FUNCTION_BLOCK Axis
//VAR_INPUT	
//END_VAR
VAR_OUTPUT
	Axis_Error			: BOOL;				// Error signal
	Axis_ErrorID		: UDINT;			// Error ID
	Axis_Moves			: BOOL;				// Status of moving
END_VAR
VAR
	// =============== Done signals MC Block =================
	JogDone			    : BOOL;					// Status of function block MC_Jog
	ResetDone		    : BOOL;					// Status of function block MC_Reset
	HaltDone		    : BOOL;					// Status of function block MC_Halt
	HomeDone		    : BOOL;					// Status of function block MC_Home
  	MoveAbsoluteDone : BOOL;        // Status of function block MC_MoveAbsolute
  	ExtSetPiontDone 	: BOOL;         		// Status of function block MC_ExtSetPointGenDisable

	// =============== Control variables ======================
	//Home_Back_Start	: BOOL;
	//Drive_Home		: BOOL;
	
	// =============== State variables ========================
	Power_StatusEnable	: BOOL;					// Enable feedback
	
	// ============= Velocity, override ,Position==============
	Velocity_Jog		: LREAL;				// Jog velocity
	Velocity_Move		: LREAL;				// Target velocity
	Velocity_Home		: LREAL;				// Home velocity
	Velocity_Absolute	: LREAL;				// MoveAbsolute velocity
	Velocity_Relative	: LREAL;				// MoveRelative velocity
	fOverride 			: LREAL := 100.0;		// Override 100%
  Home_Position   : LREAL;        // The absolute position after Home will be
	
	// =============== Trigger function blocks ================
	
	TriggerHalt	: R_TRIG;				// Trigger to recognize rising edge of halt input
	TriggerReset : R_TRIG;				// Trigger to recognize rising edge of reset input
	
	// =============== Axis reference =========================
	AxisRef			: AXIS_REF;				// Axis reference (process data plc/nc)
	
	// =============== About axis turque ====================
	Axis_Current_Turque 	: INT;
  	Axis_Max_Turque       	: INT;

	// ================= Sensor FeedBack ====================
  	Proximity_Switch      : DINT;
	
	// =============== Motion function blocks =================
	Axis_Power 			: MC_Power;				// FB for enable and override			[上电]
	Axis_Home			: MC_Home;				// FB for axis home						[找零]
	Axis_Reset 			: MC_Reset;				// FB to reset axis						[复位]
	Axis_Jog			: MC_Jog;				// FB to jog axis						[点动]
	Axis_Stop 			: MC_Stop;				// FB to stop axis						[停止]
	Axis_Halt			: MC_Halt;				// FB to halt axis						[停止]
	Axis_Move			: MC_MoveVelocity;		// FB to move axis (velocity movement)	[匀速运动]
	Axis_MoveAbsolute 	: MC_MoveAbsolute;		// FB to move axis absolutely			[绝对位置运动]
	Axis_MoveRelative	: MC_MoveRelative;		// FB to move axis relatively			[相对位置运动]
  	Axis_ActPosition  : MC_ReadActualPosition; // FB to read the actual position of axis  [读取电机轴的实际位置]
	Axis_ActVelocity	: MC_ReadActualVelocity;// FB to read the actual Velocity of axis [读取电机轴的实际速度]
	Axis_Delay			: Delay;				// FB to operate the delay program		[延迟程序]
	Axis_ExtSetPiontEnable	: MC_ExtSetPointGenEnable;	// FB to enable extsetpoint		[外部函数发生使能]
	Axis_ExtSetPiontDisable	: MC_ExtSetPointGenDisable;	// FB to disable extsetpoint	[外部函数结束使能]
  
  // =============== Timer =================
  Delay         : TON;          //[定时器]
END_VAR

PROPERTY ActPosition : LREAL
GET
Axis_ActPosition( Axis:= AxisRef, Enable:= TRUE );
ActPosition := Axis_ActPosition.Position;
END_GET
END_PROPERTY

PROPERTY ActVelocity : LREAL
GET
Axis_ActVelocity( Axis:= AxisRef, Enable:= TRUE,  ActualVelocity=> ActVelocity);
END_GET
END_PROPERTY

PROPERTY Current_Turque_Value : INT
GET
Current_Turque_Value := Axis_Current_Turque;
END_GET
SET
Axis_Current_Turque := Current_Turque_Value;
END_SET
END_PROPERTY

METHOD ExtSetPoint
VAR_INPUT
	Drive_ExtSetPointEnable 	: BOOL;		// 使能外部信号开始信号
	Drive_ExtSetPointDisable 	: BOOL;		// 使能外部信号结束信号
	ExSetPosition				: LREAL;	// 外部信号位置
	//Axis_Current_Turque 		: INT;		// 边界条件：丝杠位置到达两端卡死
END_VAR
// =======================外部信号发生程序==========================

IF NOT Axis_ExtSetPiontEnable.Error THEN
	Axis_ExtSetPiontEnable(	Axis:= AxisRef, 
							Execute:= Drive_ExtSetPointEnable, 
							Position:= ExSetPosition, 
							PositionType:= POSITIONTYPE_ABSOLUTE );
END_IF

IF Axis_ExtSetPiontEnable.Done THEN
	ExtSetPiontDone := 1;
	MC_ExtSetPointGenFeed(	Position:= ExSetPosition, 
							Velocity:= 10, 
							Acceleration:= 10, 
							Direction:= 1, 		// 1 = positive direction
							Axis:= AxisRef );
END_IF	

IF NOT Axis_ExtSetPiontDisable.Error THEN 
	Axis_ExtSetPiontDisable(	Axis:= AxisRef, 
								Execute:= Drive_ExtSetPointDisable);
END_IF
								
IF Axis_ExtSetPiontEnable.Error OR Axis_ExtSetPiontDisable.Error OR ABS(Axis_Current_Turque) > Axis_Max_Turque THEN
	IF Axis_ExtSetPiontEnable.Error OR Axis_ExtSetPiontDisable.Error THEN
		Axis_Error		:= TRUE;
		Axis_ErrorID 	:= Axis_Home.ErrorID;
	END_IF
	Axis_ExtSetPiontEnable(	Axis:= AxisRef, 
							Execute:= 0 );
	Axis_ExtSetPiontDisable(	Axis:= AxisRef, 
								Execute:= 1);
END_IF
END_METHOD

METHOD Halt : BOOL
VAR_INPUT
	DriveHalt		: BOOL;					// Request stop
END_VAR
// =======================电机运动停止程序==========================

IF DriveHalt THEN
	// Move Execute FALSE
	Axis_Move(	Execute	:= FALSE,
				Axis 	:= AxisRef);
ELSE
	// Reset done signal
	HaltDone := FALSE;
END_IF

// Trigger
TriggerHalt(CLK := DriveHalt);

IF TriggerHalt.Q THEN
	Axis_Halt(	Execute	:= TRUE,
				Axis 	:= AxisRef);
ELSE
	Axis_Halt(Axis := AxisRef);
END_IF

// Done / Error / Command aborted
IF Axis_Halt.Done OR Axis_Halt.Error OR Axis_Halt.CommandAborted THEN
	Axis_Error		:= Axis_Halt.Error;
	Axis_ErrorID 	:= Axis_Halt.ErrorID;
	HaltDone 		:= Axis_Halt.Done;
	
	Axis_Move(	Execute	:= FALSE,
				Axis 	:= AxisRef);
				
	Axis_Halt(	Execute	:= FALSE,
				Axis 	:= AxisRef);
END_IF

// =========================================================
END_METHOD

METHOD Home
VAR_INPUT
	//Back_Start 				: BOOL;
	//Velocity_Home	:LREAL;
	//Axis_Current_Turque 	: INT;
	Drive_Home				: BOOL;
END_VAR

VAR
	//HomeSet					: BOOL;
	BackDone				: BOOL;					// 电机退回到顶点位，该标志位使能
END_VAR
// =======================找零程序==========================
// 找零程序过程为：先让丝杠回退，到达机械限位后停止,并用程序将该位置置为零位

//======================丝杠回退========================
Jog_Backward(Drive_Jog_Backward:= (Drive_Home AND (NOT BackDone)));
Jog_Velocity := Velocity_Home;
HomeDone := Axis_MoveAbsolute.Done;					// 找零结束的标志为丝杠伸长到制定距离
	
IF NOT Axis_Home.Error THEN
	IF ABS(Axis_Current_Turque) > Axis_Max_Turque AND NOT BackDone THEN
		//Drive_Home :=0;
		Jog_Backward(Drive_Jog_Backward:= 0);
		Delay(IN:= NOT Delay.Q, PT:=T#200MS, Q=> , ET=> );
		Axis_Home( 	Axis:= AxisRef, 
					Execute:= Delay.Q, 
					Position:= 0, 
					HomingMode:= MC_Direct);
		BackDone := Axis_Home.Done;				
	END_IF
	IF BackDone AND Drive_Home THEN
		Move_Absolute(Drive_Move_Absolute:= TRUE, Absolute_Position:= Home_Position );
		IF Axis_MoveAbsolute.Done THEN
			BackDone := FALSE;
			Drive_Home	:= FALSE;
		END_IF
	END_IF
END_IF

(*IF HomeSet THEN
	Jog_Backward(Drive_Jog_Backward:= 0,  Axis_Current_Turque:= Axis_Current_Turque);
	HomeDone := 1;
END_IF*)

IF Axis_Home.Error OR Axis_Home.CommandAborted OR ABS(Axis_Current_Turque) < Axis_Max_Turque THEN
	IF Axis_Jog.Error THEN
		Axis_Error		:= TRUE;
		Axis_ErrorID 	:= Axis_Home.ErrorID;
	END_IF
	Axis_Home( 	Axis:= AxisRef, 
				Execute:= FALSE);
END_IF

// =========================================================
END_METHOD

PROPERTY Home_Absolute_Position : LREAL
GET
Home_Absolute_Position := Home_Position;
END_GET
SET
Home_Position := Home_Absolute_Position;
END_SET
END_PROPERTY

METHOD Home_Sensor
VAR_INPUT
	Drive_Home				: BOOL;			// 调零使能信号
	Home_Switch				: BOOL;			// 零位调零传感器信号
	//MaxPosition_Swicth		: BOOL;
END_VAR

VAR
	//HomeSet				: BOOL;
	BackDone				: BOOL;					// 电机退回到顶点位，该标志位使能
END_VAR
// =======================找零程序==========================
// 找零程序过程为：先让丝杠回退，当传感器检测到金属表面并反馈信号后, 程序将该位置置为零位

//======================丝杠回退========================
Jog_Backward(Drive_Jog_Backward:= Drive_Home);
Jog_Velocity := Velocity_Home;
HomeDone := Axis_MoveAbsolute.Done;					// 回到零点的标志为丝杠伸长到制定距离
	
IF NOT Axis_Home.Error THEN
	IF Home_Switch AND NOT HomeDone THEN
		Drive_Home :=0;
		Jog_Backward(Drive_Jog_Backward:= Drive_Home);
		Delay(IN:= NOT Delay.Q, PT:=T#200MS, Q=> , ET=> );
		Axis_Home( 	Axis:= AxisRef, 
					Execute:= Delay.Q,
					Position:= 0, 
					HomingMode:= MC_Direct);
		BackDone := Axis_Home.Done;
	END_IF
	IF BackDone THEN
		Move_Absolute(Drive_Move_Absolute:= TRUE, Absolute_Position:= 20);
		IF Axis_MoveAbsolute.Done THEN
			BackDone := FALSE;
		END_IF
	END_IF
END_IF

(*IF HomeSet THEN
	Jog_Backward(Drive_Jog_Backward:= 0,  Axis_Current_Turque:= Axis_Current_Turque);
	HomeDone := 1;
END_IF*)

IF Axis_Home.Error OR Axis_Home.CommandAborted OR ABS(Axis_Current_Turque) < Axis_Max_Turque THEN
	IF Axis_Jog.Error THEN
		Axis_Error		:= TRUE;
		Axis_ErrorID 	:= Axis_Home.ErrorID;
	END_IF
	Axis_Home( 	Axis:= AxisRef, 
				Execute:= FALSE);
END_IF

// =========================================================
END_METHOD

PROPERTY Home_Velocity : LREAL
GET
Home_Velocity := Velocity_Home;
END_GET
SET
Velocity_Home := Home_Velocity;
END_SET
END_PROPERTY

METHOD Jog_Backward
VAR_INPUT
	Drive_Jog_Backward	: BOOL;				//点动后退使能信号
	//Velocity_Jog		: LREAL;			//点动速度
	//Axis_Current_Turque : INT;				//边界条件：丝杠位置到达两端卡死
END_VAR
// =======================点动后退==========================
// 点动后退用在找零中的位置移动

IF NOT Axis_Jog.Error THEN
	Axis_Jog( 	Axis:= AxisRef, 
				JogForward:= 0, 
				JogBackwards:= Drive_Jog_Backward, 
				Mode:= MC_JOGMODE_CONTINOUS, 
				Velocity:= Velocity_Jog);
END_IF

IF Axis_Jog.Error OR Axis_Jog.CommandAborted OR ABS(Axis_Current_Turque) > Axis_Max_Turque THEN
	IF Axis_Jog.Error THEN
		Axis_Error		:= TRUE;
		Axis_ErrorID 	:= Axis_Jog.ErrorID;
	END_IF
	
	Axis_Jog(	JogForward:= 0, 
				JogBackwards:= 0, 
				Axis := AxisRef);
END_IF

(*IF ABS(Axis_Current_Turque) <1000 AND JogDone =1 THEN
	Axis_Jog(	JogForward:= 0, 
				JogBackwards:= 0, 
				Axis := AxisRef);
	JogDone :=0;
END_IF*)
				
// =========================================================
END_METHOD

METHOD Jog_Forward : BOOL
VAR_INPUT
	Drive_Jog_Forward	: BOOL;				//点动前进使能信号
	//Velocity_Jog		: LREAL;			//点动速度
	//Axis_Current_Turque : INT;				//边界条件：丝杠位置到达两端卡死
END_VAR
// =======================点动前进==========================


IF NOT Axis_Jog.Error THEN
	Axis_Jog( 	Axis:= AxisRef, 
				JogForward:= Drive_Jog_Forward, 
				JogBackwards:= 0, 
				Mode:= MC_JOGMODE_CONTINOUS, 
				Velocity:= Velocity_Jog);
END_IF

IF Axis_Jog.Error OR Axis_Jog.CommandAborted OR ABS(Axis_Current_Turque) > Axis_Max_Turque THEN
	IF Axis_Jog.Error THEN
		Axis_Error		:= TRUE;
		Axis_ErrorID 	:= Axis_Jog.ErrorID;
	END_IF
	
	Axis_Jog(	JogForward:= 0, 
				JogBackwards:= 0, 
				Axis := AxisRef);
END_IF

(*IF ABS(Axis_Current_Turque) <1000 AND JogDone =1 THEN
	Axis_Jog(	JogForward:= 0, 
				JogBackwards:= 0, 
				Axis := AxisRef);
	JogDone :=0;
END_IF*)
				
// =========================================================
END_METHOD

// =======================读写点动程序中的速度值==========================

PROPERTY Jog_Velocity : LREAL
GET
Jog_Velocity := Velocity_Jog;
END_GET
SET
Velocity_Jog := Jog_Velocity;
END_SET
END_PROPERTY

PROPERTY Max_Turque_Value : INT
SET
Axis_Max_Turque := Max_Turque_Value;
END_SET
END_PROPERTY

METHOD Move_Absolute
VAR_INPUT
	Drive_Move_Absolute : BOOL;				// 运动使能信号
	Absolute_Position	: LREAL;			// 绝对运动位置
	//Move_Velocity		: LREAL;			// 运动速度
	//Axis_Current_Turque : INT;			// 边界条件：丝杠位置到达两端卡死
END_VAR
// =======================绝对运动==========================

IF NOT Axis_MoveAbsolute.Error THEN
	Axis_MoveAbsolute(	Axis:= AxisRef, 
						Execute:= Drive_Move_Absolute, 
						Position:= Absolute_Position, 
						Velocity:= Velocity_Absolute, 
						BufferMode:= MC_Aborting );
	MoveAbsoluteDone := Axis_MoveAbsolute.Done;			// 运动到指定位置后置位
END_IF

IF Axis_MoveAbsolute.Error OR Axis_MoveAbsolute.CommandAborted OR ABS(Axis_Current_Turque) > Axis_Max_Turque THEN
	IF Axis_MoveAbsolute.Error THEN
		Axis_Error		:= TRUE;
		Axis_ErrorID 	:= Axis_MoveAbsolute.ErrorID;
	END_IF
	
	Axis_MoveAbsolute(	Axis:= AxisRef, 
						Execute:= 0, 
						BufferMode:= MC_Aborting);
END_IF

// =========================================================
END_METHOD

// =======================读写绝对运动程序中的速度值==========================

PROPERTY Move_Absolute_Velocity : LREAL
GET
Move_Absolute_Velocity := Velocity_Absolute;
END_GET
SET
Velocity_Absolute := Move_Absolute_Velocity;
END_SET
END_PROPERTY

METHOD Move_Backward
VAR_INPUT
	Move_Backward_Start : BOOL;					//匀速后退使能信号
	//Axis_Current_Turque : INT;					//边界条件：丝杠位置到达两端卡死
END_VAR
// =======================匀速后退==========================

// Not error
IF NOT Axis_Move.Error THEN
	Axis_Move(	Execute 	:= Move_Backward_Start,
				Velocity 	:= Velocity_Move,
				Direction 	:= MC_Negative_Direction,
				Axis 		:= AxisRef );
END_IF

// Error / Command aborted
IF Axis_Move.Error OR Axis_Move.CommandAborted OR ABS(Axis_Current_Turque) > Axis_Max_Turque THEN
	IF Axis_Move.Error THEN
		Axis_Error		:= TRUE;
		Axis_ErrorID 	:= Axis_Move.ErrorID;
	END_IF
	
	Axis_Move(	Execute	:= FALSE,
				Axis 	:= AxisRef);
END_IF

// =========================================================
END_METHOD

METHOD Move_Fordward
VAR_INPUT
	Move_Forward_Start : BOOL;					//匀速前进使能信号
	//Axis_Current_Turque : INT;					//边界条件：丝杠位置到达两端卡死
END_VAR
// =======================匀速前进==========================

// Not error
IF NOT Axis_Move.Error THEN
	Axis_Move(	Execute 	:= Move_Forward_Start,
				Velocity 	:= Velocity_Move,
				Direction 	:= MC_Positive_Direction,
				Axis 		:= AxisRef );
END_IF

// Error / Command aborted
IF Axis_Move.Error OR Axis_Move.CommandAborted OR ABS(Axis_Current_Turque) > Axis_Max_Turque THEN
	IF Axis_Move.Error THEN
		Axis_Error		:= TRUE;
		Axis_ErrorID 	:= Axis_Move.ErrorID;
	END_IF
	
	Axis_Move(	Execute	:= FALSE,
				Axis 	:= AxisRef);
END_IF

// =========================================================
END_METHOD

METHOD Move_Relative
VAR_INPUT
	Drive_Move_Relative		: BOOL;				// 运动使能信号
	Relative_Position		: LREAL;			// 相对运动位置
	//Move_Velocity			: LREAL;			// 运动速度
	//Axis_Current_Turque 	: INT;				// 边界条件：丝杠位置到达两端卡死
END_VAR
// =======================相对运动==========================

IF NOT Axis_MoveRelative.Error THEN
	Axis_MoveRelative(	Axis:= AxisRef, 
						Execute:= Drive_Move_Relative, 
						Distance:= Relative_Position, 
						Velocity:= Velocity_Relative, 
						BufferMode:= MC_Aborting );
END_IF

IF Axis_MoveRelative.Error OR Axis_MoveRelative.CommandAborted OR ABS(Axis_Current_Turque) > Axis_Max_Turque THEN
	IF Axis_MoveRelative.Error THEN
		Axis_Error		:= TRUE;
		Axis_ErrorID 	:= Axis_MoveRelative.ErrorID;
	END_IF
	
	Axis_MoveRelative(	Axis:= AxisRef, 
						Execute:= 0, 
						BufferMode:= MC_Aborting);
END_IF

// =========================================================
END_METHOD

// =======================读写相对运动程序中的速度值==========================

PROPERTY Move_Relative_Velocity : LREAL
GET
Move_Relative_Velocity := Velocity_Relative;
END_GET
SET
Velocity_Relative := Move_Relative_Velocity;
END_SET
END_PROPERTY

PROPERTY Move_Velocity : LREAL
GET
Move_Velocity := Velocity_Move;
END_GET
SET
Velocity_Move :=Move_Velocity :=10;
END_SET
END_PROPERTY

METHOD Power
VAR_INPUT
	Axis_Enable : BOOL;
END_VAR
// =======================上电程序==========================

Axis_Power(	Enable 			:= Axis_Enable, 
			Enable_Positive	:= Axis_Enable, 
			Enable_Negative	:= Axis_Enable, 
			Override		:= fOverride,
			Axis			:= AxisRef,
			Status			=> Power_StatusEnable);
			
IF Axis_Power.Error THEN
	Axis_Error		:= TRUE;
	Axis_ErrorID 	:= Axis_Power.ErrorID;
END_IF

AxisRef.ReadStatus();

Axis_Moves := AxisRef.Status.Moving;

// ==========================================================
END_METHOD

METHOD Reset
VAR_INPUT
	Drive_Reset		: BOOL;					// Request reset
END_VAR
// =====================驱动重置程序==========================

IF NOT Drive_Reset THEN
	ResetDone 	:= FALSE;
END_IF

// Trigger(触发器)
TriggerReset(CLK := Drive_Reset);

IF TriggerReset.Q THEN
	HaltDone 	:= FALSE;
	
	Axis_Reset(Execute := TRUE, Axis := AxisRef);
ELSE
	Axis_Reset(Axis := AxisRef);
END_IF

// Done / Error
IF Axis_Reset.Done OR Axis_Reset.Error THEN
	Axis_Error		:= Axis_Reset.Error;
	Axis_ErrorID 	:= Axis_Reset.ErrorID;
	ResetDone 		:= Axis_Reset.Done;

	Axis_Reset(	Execute	:= FALSE, Axis 	:= AxisRef);
END_IF

// =========================================================
END_METHOD

PROPERTY State_ExtSetPiontDone : BOOL
GET
State_ExtSetPiontDone := ExtSetPiontDone;
END_GET
END_PROPERTY

// =======================回零结束信号==========================

PROPERTY State_HomeDone : BOOL
GET
State_HomeDone := HomeDone;
END_GET
END_PROPERTY

// =======================点动结束信号==========================

PROPERTY State_JogDone : BOOL
GET
State_JogDone := JogDone;
END_GET
END_PROPERTY

PROPERTY State_MoveAbsoluteDone : BOOL
GET
State_MoveAbsoluteDone := MoveAbsoluteDone;
END_GET
END_PROPERTY

// =======================上电状态信号==========================

PROPERTY State_PowerStatus : BOOL
GET
State_PowerStatus := Power_StatusEnable;
END_GET
END_PROPERTY

// =======================复位结束信号==========================

PROPERTY State_ResetDone : BOOL
GET
State_ResetDone := ResetDone;
END_GET
END_PROPERTY

END_FUNCTION_BLOCK

(* stored: Version 1.1.0.1, ProductVersion 3.1.4020.12
   POU Axis: Id {875f83f1-eb97-483f-b7d6-014637e061f1}, SpecialFunc None
   Property ActPosition: Id {3015e613-88a6-44b7-bfd3-2c06df6f075d}
   Get Get: Id {49f49f46-670a-4f33-894d-6ca9ed093408}
   Property ActVelocity: Id {6ba788af-13d6-45aa-88b8-c4b15f3b7302}
   Get Get: Id {d9e77e56-00f7-4ebc-9fc8-803356b7adfe}
   Property Current_Turque_Value: Id {3a2f771d-3376-4640-bd97-650af6e34455}
   Get Get: Id {c1b780dc-fdc4-4a6a-9032-d0ef9263bab2}
   Set Set: Id {51333a67-cd8e-4eac-b9a4-9ecae4706b9e}
   Method ExtSetPoint: Id {e3dd3d6b-d150-49a2-a8d7-a7990a606e4c}
   Method Halt: Id {d7ff254f-2dd7-462f-bdbd-9197c2ffdaa3}
   Method Home: Id {313e1eef-e597-492a-a006-a8453e584cfd}
   Property Home_Absolute_Position: Id {4b2bc104-de65-4853-bc96-2381d638aa2c}
   Get Get: Id {b2452760-cdc1-4500-a807-21088ae1fa11}
   Set Set: Id {13130e40-cbc6-42ec-8c48-c9869e4c03d4}
   Method Home_Sensor: Id {a22704a8-b010-4cc1-be73-1967f40884b9}
   Property Home_Velocity: Id {075d0823-6614-4698-9d00-5a9266b58e8c}
   Get Get: Id {41764938-04f0-496d-b0d3-2075d0bf01de}
   Set Set: Id {81d43709-9b51-4423-8fa5-968a12b8eb76}
   Method Jog_Backward: Id {99d13956-4937-48a4-92d1-297e5120f462}
   Method Jog_Forward: Id {9deceb4f-22e3-43d3-abba-cc65da0a988f}
   Property Jog_Velocity: Id {fbf70f23-ccbc-42f7-9290-364343308531}
   Get Get: Id {43fe7bb4-cb6d-421c-bc16-b82658b77bde}
   Set Set: Id {5232cb37-92d1-44d0-9e06-54bf215c7cbc}
   Property Max_Turque_Value: Id {c8624b49-e9f6-4c92-b644-367354523826}
   Set Set: Id {61f18c04-0a46-4043-b21d-3c09633e0ec4}
   Method Move_Absolute: Id {90058d1c-d052-4ccf-9289-5faf8ddb84ca}
   Property Move_Absolute_Velocity: Id {7cb9ac45-b7a3-4012-b6de-6d6ce49b5a54}
   Get Get: Id {72f69858-955f-443c-af51-259e8e609d4c}
   Set Set: Id {c5a5a778-30ed-4aa2-a2ed-0d898d7d6498}
   Method Move_Backward: Id {d07db03f-d706-432b-92a0-251009b4d606}
   Method Move_Fordward: Id {30d70636-f830-44c4-adf2-54f90ee067a6}
   Method Move_Relative: Id {7b541efd-c3a2-463f-9025-d3f3cd116050}
   Property Move_Relative_Velocity: Id {10d568b7-1224-4f3c-82dc-f2b473343afd}
   Get Get: Id {2ef19610-9237-4e3e-8453-be0ff288ee9e}
   Set Set: Id {333783a0-b8e9-41f4-b7a2-5d9a70341bc4}
   Property Move_Velocity: Id {21dc1ad2-a805-4cc5-ba52-5eb4a3378ad2}
   Get Get: Id {febdf6e5-1449-4037-ae17-7b2213508e1c}
   Set Set: Id {44a4395c-73de-4ae0-b7b0-c7902df3efbf}
   Method Power: Id {cc0985ad-b04b-4e99-b924-c7a9a3e5739c}
   Method Reset: Id {dedc8057-c4ab-4248-b14b-274fa3c9288f}
   Property State_ExtSetPiontDone: Id {6243132d-fdac-4a44-aabc-1626db2c504e}
   Get Get: Id {c75a34d6-3b40-4dd5-b205-992b19da25da}
   Property State_HomeDone: Id {b05cc381-4a45-4536-92f9-829385d416fe}
   Get Get: Id {61dc4a9a-ce60-4f15-af37-592d6a63af40}
   Property State_JogDone: Id {3c0f115e-f80a-44b9-a70e-39bb83e64c81}
   Get Get: Id {19bafe7b-2de8-400b-a26d-d4ad9918869f}
   Property State_MoveAbsoluteDone: Id {7b7a8b76-a437-47fb-99a9-6a9d632d1395}
   Get Get: Id {15c8003a-8e08-4231-b9e8-509a81a20964}
   Property State_PowerStatus: Id {26f2d544-ee3f-4b26-afb9-71118906e7d1}
   Get Get: Id {d3af8348-880a-4df8-b9de-20b9d23a495b}
   Property State_ResetDone: Id {e8bc9f4f-5bd7-4f76-a8c5-8b726ec5b1c8}
   Get Get: Id {6d6b999c-0bec-46b0-8fb1-c5d8586fb5ed} *)
